// TwinCAT 3 PLC project ModbusPlc
// Title: ModbusPlc
// Company: MyLovelyCompany
// Author: PTKu
// ProjectVersion: 0.0.0.1
// ProgramVersion: 3.1.4023.0
// libraries:
//   Tc2_Standard, * (Beckhoff Automation GmbH)
//   Tc2_System, * (Beckhoff Automation GmbH)
//   Tc3_Module, * (Beckhoff Automation GmbH)
//   TcoCore, 0.4.2.560 (Vortex.Library)
// project tree:
//   / PlcTask.TcTTO
//   POUs/ ModBusContext.TcPOU, MAIN.TcPOU
// real-time tasks:
//   TASK PlcTask: cycle T#10ms, priority 20, ADS port 350

CONFIGURATION ModbusPlc
    RESOURCE PLC ON TwinCAT3
        TASK PlcTask(INTERVAL := T#10ms, PRIORITY := 20);
        PROGRAM MAIN WITH PlcTask : MAIN;
    END_RESOURCE
END_CONFIGURATION

// ---- POUs/MAIN.TcPOU
PROGRAM MAIN
VAR
	// More about context and tasks here: https://docs.tcopengroup.org/articles/TcOpenFramework/application.html
	_context : ModBusContext;
END_VAR

// This runs the context.
_context.Run();

END_PROGRAM

// ---- POUs/ModBusContext.TcPOU
FUNCTION_BLOCK ModBusContext EXTENDS TcoCore.TcoContext
VAR
	// Remote task
	_touchModbus : TcoCore.TcoRemoteTask(THIS^);  
END_VAR

VAR
	// Accessing these variables.
	modbusvar1 : INT;
	modbusvar2 : INT;
END_VAR

(*~
	<docu>
		<summary>
			Main method of the TcoContext. This is the entry point of any control logic that belongs to this context. 
			The call of this method is ensured by calling the <c>InstanceName.Run()</c> method, and it must not be called explicitly.
			This method is abstract, and it must be overridden in derived block.
		</summary>
	</docu>
~*)
METHOD PROTECTED  Main
// Invoke fires the execution of C# code handling ModBus communication
IF(_touchModbus.Invoke().Done OR _touchModbus.Error) THEN
	// When done or failure this kicks the remote call again.
	_touchModbus.Restore();	
END_IF

// You just need to call this...
_touchModbus();
END_METHOD

END_FUNCTION_BLOCK
